Yaskawa INFORM job: MAINTENANCE-POSITION.JBI

/JOB
//NAME MAINTENANCE-POSITION
//POS
///NPOS 1,1,0,0,0,0
///TOOL 0
///POSTYPE PULSE
///PULSE
C00000=2,0,-2,1,0,46844
BC00000=175236
//INST
///DATE 2018/08/27 15:17
///ATTR SC,RW
///GROUP1 RB1,BS1
NOP
MOVJ C00000 BC00000 VJ=5.00
END
